// Mitsubishi GX Works2 project: ArielKing4.12   PLC: FX3G

// global labels: Global1
VAR_GLOBAL
  Start_Day AT X007 : BOOL;
  Emergency AT X005 : BOOL;
  Check_Products AT M1 : BOOL;
  Work_Day_On AT Y000 : BOOL;
  Start_Blend AT X003 : BOOL;
  Shibulet_Amount AT D1102 : INT;
END_VAR
VAR_GLOBAL CONSTANT
  GE_Eth_Connection_Status : INT := 400;
  GE_Eth_k0 : INT := 400;
  GE_Eth_k400 : REAL := 400;
  GE_Eth_k320 : REAL := 320;
  GE_Eth_k160 : REAL := 160;
END_VAR
VAR_GLOBAL
  Analog_Input_1 AT D8280 : INT;
END_VAR
VAR_GLOBAL CONSTANT
  GE_Eth_K5 : INT := 400;
  LE_Eth_K5 : REAL := 5;
  GT_Eth_K5 : REAL := 5;
END_VAR
VAR_GLOBAL
  Protein AT M3 : BOOL;
  Classy AT M4 : BOOL;
END_VAR
VAR_GLOBAL CONSTANT
  SUB_Eth_1k240 : INT := 400;
  LT_Eth_k320 : REAL := 320;
  LT_Eth_k160 : REAL := 160;
  LT_Eth_K400 : REAL := 400;
  LT_Eth_k120 : REAL := 120;
  SUB_Eth_k240 : REAL := 240;
  SUB_Eth_k320 : REAL := 320;
  SUB_Eth_k160 : REAL := 160;
  SUB_Eth_k400 : REAL := 400;
  SUB_Eth_k120 : REAL := 120;
END_VAR
VAR_GLOBAL
  FiveS_Light AT Y003 : BOOL;
  Start_Baking AT X002 : BOOL;
  Start_Packing AT X006 : BOOL;
  TIMER1 AT TC1 : BOOL;
END_VAR
VAR_GLOBAL CONSTANT
  CONST5 : INT := 50;
END_VAR
VAR_GLOBAL
  counterBit AT TS1 : BOOL;
  GE1 : BOOL;
  GE2 : BOOL;
  GE3 : BOOL;
  LT2 : BOOL;
  GT_4 : BOOL;
  GT_5 : BOOL;
  LT3 : BOOL;
  LT1 : BOOL;
  LT6 : BOOL;
  LT4 : BOOL;
  LT5 : BOOL;
  Timer_On_5 AT M6 : BOOL;
  Iinput_Shibolet AT D1100 : REAL;
  Sibolet_Amount AT D1102 : REAL;
  Input_Protein AT D1104 : REAL;
  Input_Honey AT D1108 : REAL;
  Honey_Amount AT D1110 : REAL;
  Shibolet_Amount AT D1102 : REAL;
  Save_Analog_Value AT D8201 : REAL;
  Protein_Amount AT D1106 : REAL;
  One_Time_Restart AT CC0 : BOOL;
  Check_Product_Shibolet AT M10 : BOOL;
  Check_Product_Protein AT M20 : BOOL;
  Check_Product_Honey AT M30 : BOOL;
END_VAR
VAR_GLOBAL CONSTANT
  LT_Eth_K240 : REAL := 240;
END_VAR
VAR_GLOBAL
  M_0 AT M0 : BOOL;
  Y_1 AT Y001 : BOOL;
  Y_2 AT Y002 : BOOL;
  TC_2 AT TC2 : BOOL;
END_VAR
VAR_GLOBAL CONSTANT
  Twinkle_time : INT := 10;
END_VAR
VAR_GLOBAL
  TS_2 AT TS2 : BOOL;
  TC_3 AT TC3 : BOOL;
  TS_3 AT TS3 : BOOL;
  TC_4 AT TC4 : BOOL;
  TC_5 AT TC5 : BOOL;
  TS_4 AT TS4 : BOOL;
  TS_5 AT TS5 : BOOL;
END_VAR
VAR_GLOBAL CONSTANT
  Classy_Baking_time : INT := 40;
  Protein_Baking_time : INT := 50;
END_VAR
VAR_GLOBAL
  Twinkle_Stop AT M40 : BOOL;
END_VAR
VAR_GLOBAL CONSTANT
  Divide400 : REAL := 400;
END_VAR
VAR_GLOBAL
  FiveSecBlendLight AT M8 : BOOL;
  Single_Packing AT X000 : BOOL;
  One_Time_Restart1 AT CC0 : BOOL;
END_VAR
VAR_GLOBAL CONSTANT
  Check1 : WORD := 1;
END_VAR
VAR_GLOBAL
  Close_Reset_1 AT CS0 : BOOL;
  Packing_Begin AT M18 : BOOL;
  First_Snack AT CC2 : BOOL;
  Full_Package AT CC3 : BOOL;
  First_Snack_On AT CS2 : BOOL;
  Full_Package_On AT CS3 : BOOL;
  After_First_Till_Last AT Y004 : BOOL;
  Finish_Packing AT M14 : BOOL;
END_VAR
VAR_GLOBAL CONSTANT
  Add_Package : INT := 1;
  Count1 : INT := 1;
  Count8 : INT := 8;
  Add_one_pack : REAL := 1;
END_VAR
VAR_GLOBAL
  Check_Blend_Finish AT M22 : BOOL;
END_VAR
VAR_GLOBAL CONSTANT
  Make_Esroni : REAL := 10;
  Costant400 : REAL := 400;
END_VAR
VAR_GLOBAL
  Package_Amount AT D1120 : REAL;
  Analog_Output AT D8282 : INT;
END_VAR

// task Task_01 (event TRUE, interval 0, priority 31): POU_01

PROGRAM POU_01
(* structured ladder/FBD written out as ST: instructions are called as NAME(EN, inputs, outputs); _pN, _eN, _tN stand for wires *)
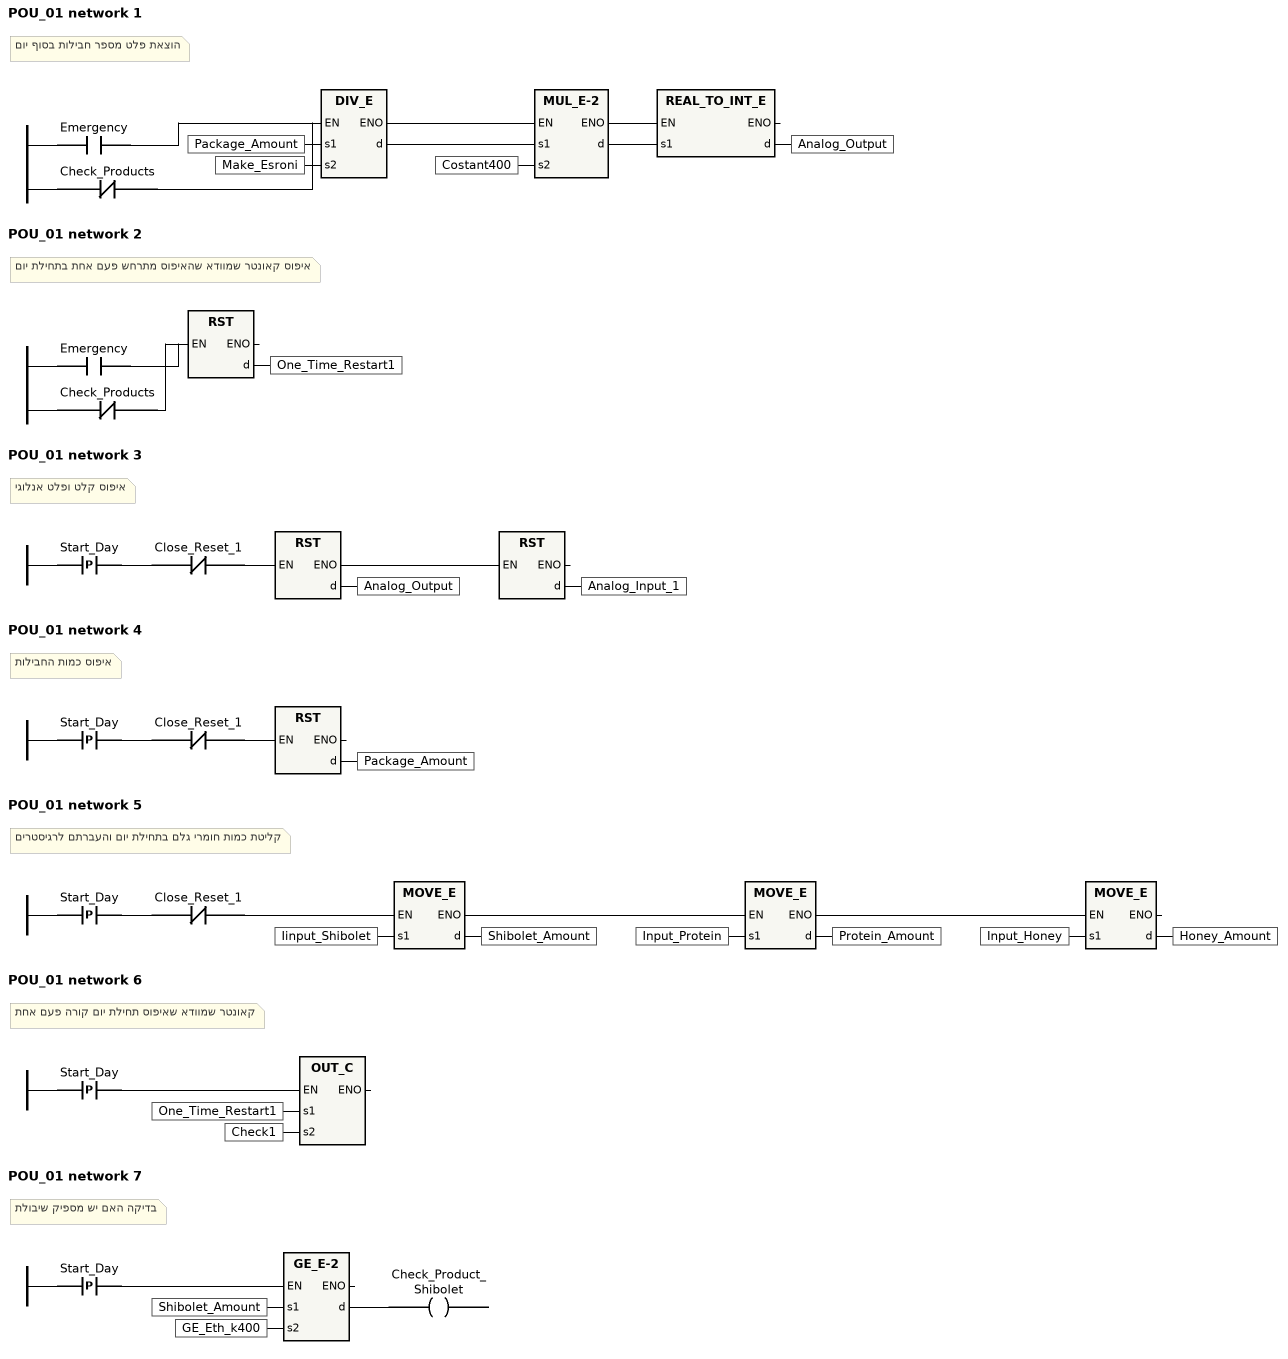
(* network 1 *)
(* הוצאת פלט מספר חבילות בסוף יום *)
_e2 := DIV_E(Emergency OR (NOT Check_Products), Package_Amount, Make_Esroni, _t1);
_e4 := MUL_E(_e2, _t1, Costant400, _t3);
REAL_TO_INT_E(_e4, _t3, Analog_Output);
(* network 2 *)
(* איפוס קאונטר שמוודא שהאיפוס מתרחש פעם אחת בתחילת יום *)
RST(Emergency OR (NOT Check_Products), One_Time_Restart1);
(* network 3 *)
(* איפוס קלט ופלט אנלוגי *)
_e1 := RST(LDP(TRUE, Start_Day) AND NOT Close_Reset_1, Analog_Output);
RST(_e1, Analog_Input_1);
(* network 4 *)
(* איפוס כמות החבילות *)
RST(LDP(TRUE, Start_Day) AND NOT Close_Reset_1, Package_Amount);
(* network 5 *)
(* קליטת כמות חומרי גלם בתחילת יום והעברתם לרגיסטרים *)
_e1 := MOVE_E(LDP(TRUE, Start_Day) AND NOT Close_Reset_1, Iinput_Shibolet, Shibolet_Amount);
_e2 := MOVE_E(_e1, Input_Protein, Protein_Amount);
MOVE_E(_e2, Input_Honey, Honey_Amount);
(* network 6 *)
(* קאונטר שמוודא שאיפוס תחילת יום קורה פעם אחת *)
OUT_C(LDP(TRUE, Start_Day), One_Time_Restart1, Check1);
(* network 7 *)
(* בדיקה האם יש מספיק שיבולת *)
GE_E(LDP(TRUE, Start_Day), Shibolet_Amount, GE_Eth_k400, _t1);
Check_Product_Shibolet := _t1;
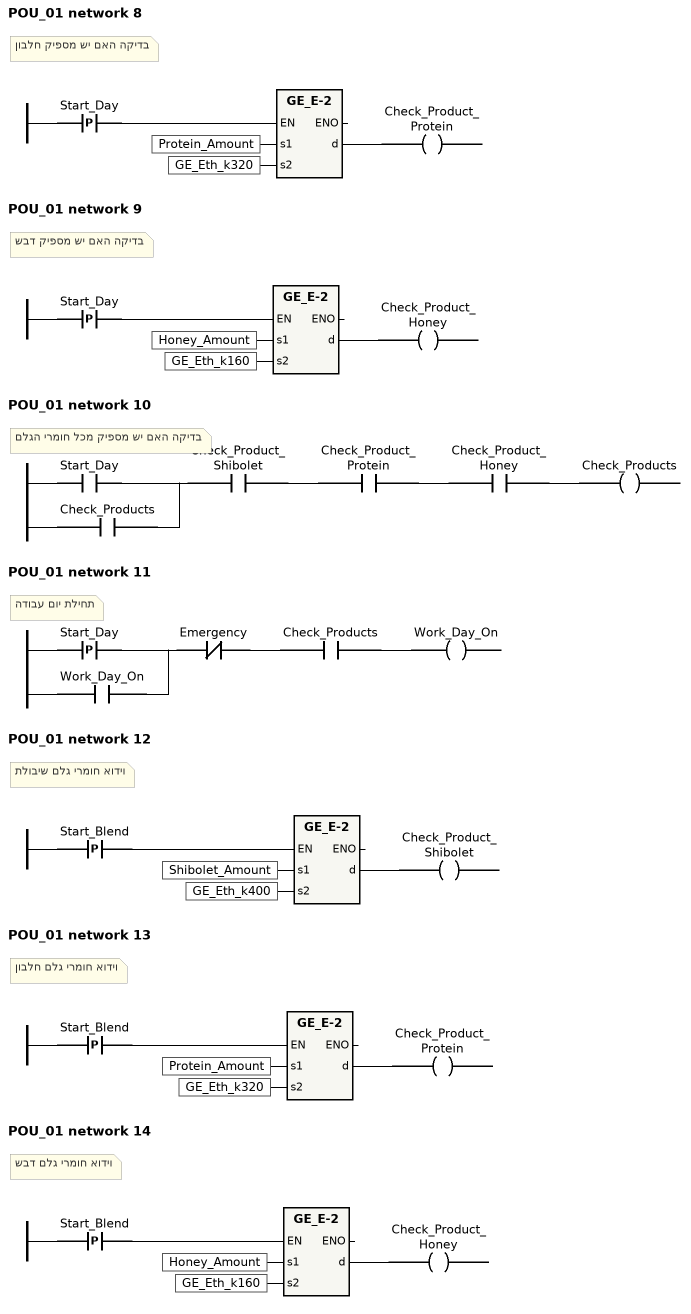
(* network 8 *)
(* בדיקה האם יש מספיק חלבון *)
GE_E(LDP(TRUE, Start_Day), Protein_Amount, GE_Eth_k320, _t1);
Check_Product_Protein := _t1;
(* network 9 *)
(* בדיקה האם יש מספיק דבש *)
GE_E(LDP(TRUE, Start_Day), Honey_Amount, GE_Eth_k160, _t1);
Check_Product_Honey := _t1;
(* network 10 *)
(* בדיקה האם יש מספיק מכל חומרי הגלם *)
Check_Products := (((Start_Day OR Check_Products) AND Check_Product_Shibolet) AND Check_Product_Protein) AND Check_Product_Honey;
(* network 11 *)
(* תחילת יום עבודה *)
Work_Day_On := ((LDP(TRUE, Start_Day) OR Work_Day_On) AND NOT Emergency) AND Check_Products;
(* network 12 *)
(* וידוא חומרי גלם שיבולת *)
GE_E(LDP(TRUE, Start_Blend), Shibolet_Amount, GE_Eth_k400, _t1);
Check_Product_Shibolet := _t1;
(* network 13 *)
(* וידוא חומרי גלם חלבון *)
GE_E(LDP(TRUE, Start_Blend), Protein_Amount, GE_Eth_k320, _t1);
Check_Product_Protein := _t1;
(* network 14 *)
(* וידוא חומרי גלם דבש *)
GE_E(LDP(TRUE, Start_Blend), Honey_Amount, GE_Eth_k160, _t1);
Check_Product_Honey := _t1;
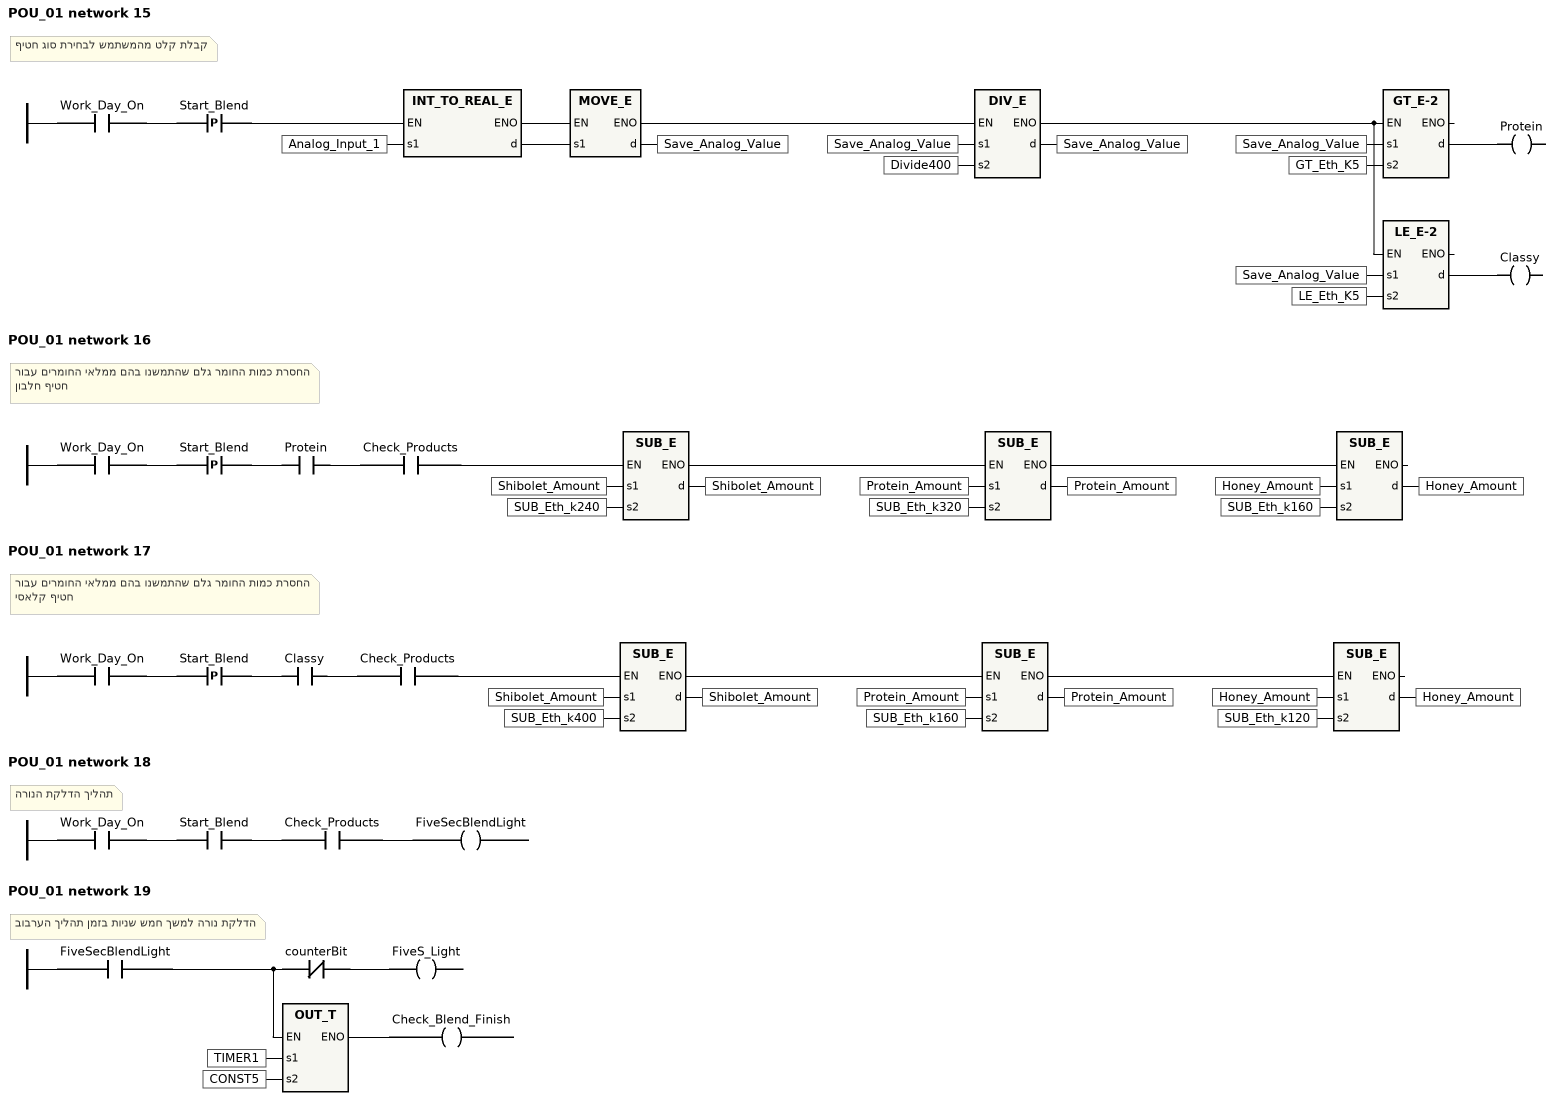
(* network 15 *)
(* קבלת קלט מהמשתמש לבחירת סוג חטיף *)
_e2 := INT_TO_REAL_E(Work_Day_On AND LDP(TRUE, Start_Blend), Analog_Input_1, _t1);
_e3 := MOVE_E(_e2, _t1, Save_Analog_Value);
_e4 := DIV_E(_e3, Save_Analog_Value, Divide400, Save_Analog_Value);
GT_E(_e4, Save_Analog_Value, GT_Eth_K5, _t5);
Protein := _t5;
LE_E(_e4, Save_Analog_Value, LE_Eth_K5, _t6);
Classy := _t6;
(* network 16 *)
(* החסרת כמות החומר גלם שהתמשנו בהם ממלאי החומרים עבור חטיף חלבון *)
_e1 := SUB_E(Work_Day_On AND LDP(TRUE, Start_Blend) AND Protein AND Check_Products, Shibolet_Amount, SUB_Eth_k240, Shibolet_Amount);
_e2 := SUB_E(_e1, Protein_Amount, SUB_Eth_k320, Protein_Amount);
SUB_E(_e2, Honey_Amount, SUB_Eth_k160, Honey_Amount);
(* network 17 *)
(* החסרת כמות החומר גלם שהתמשנו בהם ממלאי החומרים עבור חטיף קלאסי *)
_e1 := SUB_E(Work_Day_On AND LDP(TRUE, Start_Blend) AND Classy AND Check_Products, Shibolet_Amount, SUB_Eth_k400, Shibolet_Amount);
_e2 := SUB_E(_e1, Protein_Amount, SUB_Eth_k160, Protein_Amount);
SUB_E(_e2, Honey_Amount, SUB_Eth_k120, Honey_Amount);
(* network 18 *)
(* תהליך הדלקת הנורה *)
FiveSecBlendLight := Work_Day_On AND Start_Blend AND Check_Products;
(* network 19 *)
(* הדלקת נורה למשך חמש שניות בזמן תהליך הערבוב *)
FiveS_Light := FiveSecBlendLight AND NOT counterBit;
_e1 := OUT_T(FiveSecBlendLight, TIMER1, CONST5);
Check_Blend_Finish := _e1;
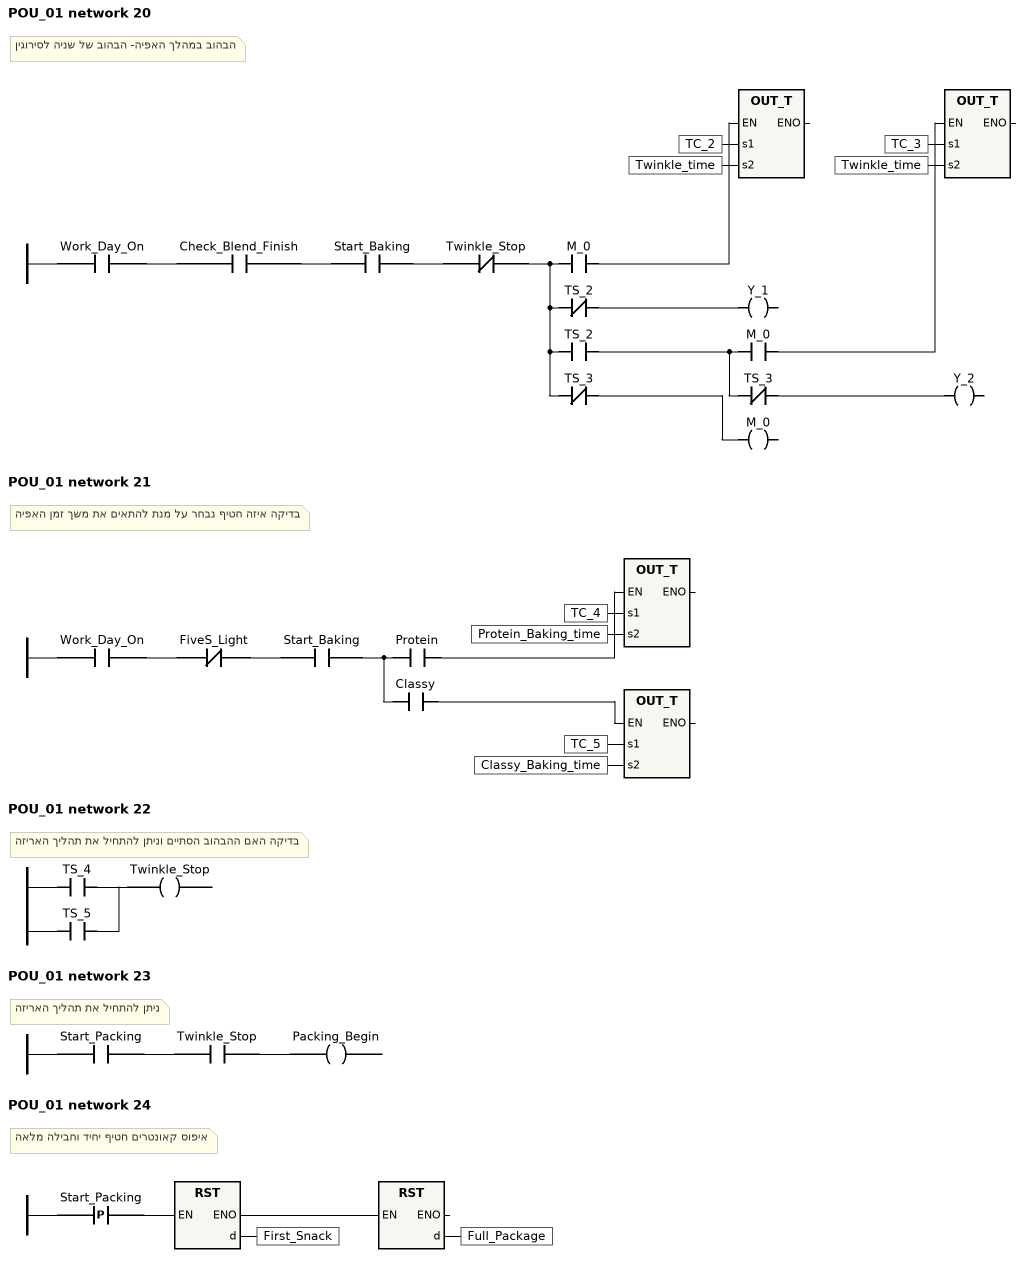
(* network 20 *)
(* הבהוב במהלך האפיה- הבהוב של שניה לסירוגין *)
_p1 := Work_Day_On AND Check_Blend_Finish AND Start_Baking AND NOT Twinkle_Stop;
OUT_T(_p1 AND M_0, TC_2, Twinkle_time);
Y_1 := _p1 AND NOT TS_2;
_p2 := _p1 AND TS_2;
OUT_T(_p2 AND M_0, TC_3, Twinkle_time);
Y_2 := _p2 AND NOT TS_3;
M_0 := _p1 AND NOT TS_3;
(* network 21 *)
(* בדיקה איזה חטיף נבחר על מנת להתאים את משך זמן האפיה *)
_p1 := Work_Day_On AND NOT FiveS_Light AND Start_Baking;
OUT_T(_p1 AND Protein, TC_4, Protein_Baking_time);
OUT_T(_p1 AND Classy, TC_5, Classy_Baking_time);
(* network 22 *)
(* בדיקה האם ההבהוב הסתיים וניתן להתחיל את תהליך האריזה *)
Twinkle_Stop := TS_4 OR TS_5;
(* network 23 *)
(* ניתן להתחיל את תהליך האריזה *)
Packing_Begin := Start_Packing AND Twinkle_Stop;
(* network 24 *)
(* איפוס קאונטרים חטיף יחיד וחבילה מלאה *)
_e1 := RST(LDP(TRUE, Start_Packing), First_Snack);
RST(_e1, Full_Package);
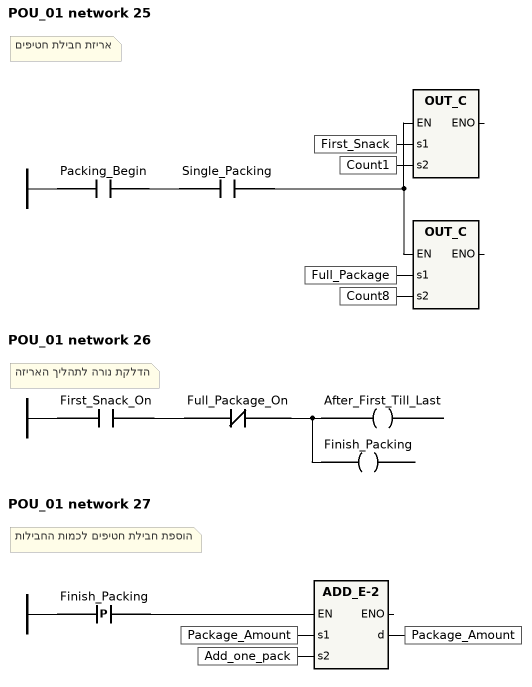
(* network 25 *)
(* אריזת חבילת חטיפים *)
_p1 := Packing_Begin AND Single_Packing;
OUT_C(_p1, First_Snack, Count1);
OUT_C(_p1, Full_Package, Count8);
(* network 26 *)
(* הדלקת נורה לתהליך האריזה *)
_p1 := First_Snack_On AND NOT Full_Package_On;
After_First_Till_Last := _p1;
Finish_Packing := _p1;
(* network 27 *)
(* הוספת חבילת חטיפים לכמות החבילות *)
ADD_E(LDP(TRUE, Finish_Packing), Package_Amount, Add_one_pack, Package_Amount);
END_PROGRAM
